(* IEC 61131-3 sources: Word/plc-course/07-timers/labs/solutions, 5 files *)

(* ---- 07-1-star-delta.st ---- *)
(* Lab 07-1: Star-delta starter.
   Module 07 (Timers). REFERENCE SOLUTION - try the lab yourself first.

   Sequence: Start -> main + star contactors on -> after StarTime the star
   contactor opens -> 100 ms dead time -> delta contactor closes.
   Training exercise only: a real starter also has hard-wired electrical and
   mechanical interlocks between the star and delta contactors. *)

PROGRAM StarDelta
  VAR (* I/O *)
    StartPB       AT %IX0.0 : BOOL;  (* Start push-button, NO: TRUE while pressed *)
    StopPB_NC     AT %IX0.1 : BOOL;  (* Stop push-button, NC: TRUE while NOT pressed *)
    OverloadOK_NC AT %IX0.2 : BOOL;  (* Overload relay contact, NC: TRUE while healthy *)
    MainK         AT %QX0.0 : BOOL;  (* Main (line) contactor *)
    StarK         AT %QX0.1 : BOOL;  (* Star contactor *)
    DeltaK        AT %QX0.2 : BOOL;  (* Delta contactor *)
  END_VAR
  VAR (* settings, e.g. written from an HMI *)
    StarTime : TIME := T#5s;         (* how long the motor starts in star *)
  END_VAR
  VAR (* internal *)
    StarTimer : TON;                 (* times the star period *)
    GapTimer  : TON;                 (* changeover dead time, star off -> delta on *)
  END_VAR

  (* 1. Run latch. The main contactor seals itself in. Stop and the overload
        both break the seal, so releasing Stop or resetting the overload relay
        can never restart the motor on its own. *)
  MainK := (StartPB OR MainK) AND StopPB_NC AND OverloadOK_NC;

  (* 2. Star period. The timer runs while the main contactor is on and is
        reset as soon as it drops out, so every new start gets a full star
        period. The timer is called on every scan, never inside an IF. *)
  StarTimer(IN := MainK, PT := StarTime);
  StarK := MainK AND NOT StarTimer.Q;

  (* 3. Changeover gap. StarTimer.Q is TRUE from the scan in which the star
        contactor is switched off, so GapTimer measures how long star has been
        off. Delta may close only after 100 ms, when the star contactor has
        had time to open and its arc to clear. *)
  GapTimer(IN := StarTimer.Q, PT := T#100ms);

  (* 4. Delta, with a software interlock against star as a second line of
        defence (the first line is the hard-wired interlock in the panel). *)
  DeltaK := MainK AND GapTimer.Q AND NOT StarK;
END_PROGRAM

CONFIGURATION Config0
  RESOURCE Res0 ON PLC
    TASK MainTask(INTERVAL := T#10ms, PRIORITY := 0);
    PROGRAM Inst0 WITH MainTask : StarDelta;
  END_RESOURCE
END_CONFIGURATION

(* ---- 07-2-flasher-beacon.st ---- *)
(* Lab 07-2: Flasher beacon with separate on and off times.
   Module 07 (Timers). REFERENCE SOLUTION - try the lab yourself first.

   Two timers that reset each other form an oscillator:
     OnTimer  times the ON phase  (beacon lit while it is timing),
     OffTimer times the OFF phase (started when OnTimer is done).
   When OffTimer is done, OnTimer's IN goes FALSE for one scan. That resets
   both timers and the cycle starts again with a new ON phase. *)

PROGRAM FlasherBeacon
  VAR (* I/O *)
    Enable AT %IX0.0 : BOOL;   (* flash request, e.g. "machine about to start" *)
    Beacon AT %QX0.0 : BOOL;   (* beacon lamp *)
  END_VAR
  VAR (* settings, e.g. written from an HMI *)
    OnTime  : TIME := T#500ms; (* lamp on time *)
    OffTime : TIME := T#1s;    (* lamp off time *)
  END_VAR
  VAR (* internal *)
    OnTimer  : TON;            (* ON phase *)
    OffTimer : TON;            (* OFF phase *)
  END_VAR

  (* ON phase: runs while enabled, until the OFF phase has finished.
     Removing Enable resets it, so the next enable starts with a full
     ON phase. *)
  OnTimer(IN := Enable AND NOT OffTimer.Q, PT := OnTime);

  (* OFF phase: starts when the ON phase is done. *)
  OffTimer(IN := OnTimer.Q, PT := OffTime);

  (* The lamp is lit while enabled and the ON phase is not yet done. *)
  Beacon := Enable AND NOT OnTimer.Q;
END_PROGRAM

CONFIGURATION Config0
  RESOURCE Res0 ON PLC
    TASK MainTask(INTERVAL := T#10ms, PRIORITY := 0);
    PROGRAM Inst0 WITH MainTask : FlasherBeacon;
  END_RESOURCE
END_CONFIGURATION

(* ---- 07-3-feedback-timeout.st ---- *)
(* Lab 07-3: Motor with run-feedback monitoring.
   Module 07 (Timers). REFERENCE SOLUTION - try the lab yourself first.

   Two supervision timers compare what we ASK the motor to do (MotorRun)
   with what it REPORTS (RunFbk):
     - fail to start: no feedback within StartTimeout of the start,
     - feedback lost: feedback was proven, then missing for LossDelay.
   A fault latches, stops the motor, and can be reset only while the run
   command is off, so a reset can never restart the motor by surprise. *)

PROGRAM FeedbackTimeout
  VAR (* I/O *)
    RunCmd    AT %IX0.0 : BOOL;  (* run request (maintained), TRUE = run *)
    RunFbk    AT %IX0.1 : BOOL;  (* running feedback: contactor aux contact or drive "running" *)
    ResetPB   AT %IX0.2 : BOOL;  (* fault reset push-button, NO *)
    MotorRun  AT %QX0.0 : BOOL;  (* contactor coil / drive run command *)
    FaultLamp AT %QX0.1 : BOOL;  (* fault lamp: on while any fault is latched *)
  END_VAR
  VAR (* settings *)
    StartTimeout : TIME := T#3s;     (* time allowed for feedback after a start *)
    LossDelay    : TIME := T#500ms;  (* feedback dropout tolerated while running *)
  END_VAR
  VAR (* alarms for the HMI *)
    FailToStart : BOOL;          (* latched: no feedback after starting *)
    FbkLost     : BOOL;          (* latched: feedback lost while running *)
  END_VAR
  VAR (* internal *)
    Proven     : BOOL;           (* feedback has been seen during this run *)
    StartTimer : TON;            (* supervises the start *)
    LossTimer  : TON;            (* supervises the running motor *)
  END_VAR

  (* 1. "Proven" remembers that feedback arrived during the current run.
        It is cleared whenever the motor is not being commanded, so every new
        start is supervised by the start timer again. MotorRun here is the
        value written at the end of the previous scan. *)
  IF NOT MotorRun THEN
    Proven := FALSE;
  ELSIF RunFbk THEN
    Proven := TRUE;
  END_IF;

  (* 2. Supervision timers. Both are called on every scan; their IN
        conditions decide when they time. *)
  StartTimer(IN := MotorRun AND NOT Proven, PT := StartTimeout);
  LossTimer(IN := MotorRun AND Proven AND NOT RunFbk, PT := LossDelay);

  (* 3. Latch the faults. *)
  IF StartTimer.Q THEN
    FailToStart := TRUE;
  END_IF;
  IF LossTimer.Q THEN
    FbkLost := TRUE;
  END_IF;

  (* 4. Reset, accepted only while the run command is off. *)
  IF ResetPB AND NOT RunCmd THEN
    FailToStart := FALSE;
    FbkLost := FALSE;
  END_IF;

  (* 5. Outputs. *)
  FaultLamp := FailToStart OR FbkLost;
  MotorRun := RunCmd AND NOT FaultLamp;
END_PROGRAM

CONFIGURATION Config0
  RESOURCE Res0 ON PLC
    TASK MainTask(INTERVAL := T#10ms, PRIORITY := 0);
    PROGRAM Inst0 WITH MainTask : FeedbackTimeout;
  END_RESOURCE
END_CONFIGURATION

(* ---- 07-4-run-hours.st ---- *)
(* Lab 07-4: Accumulating run-hours meter.
   Module 07 (Timers). REFERENCE SOLUTION - try the lab yourself first.

   Idea: use a TON purely as a stopwatch. Its ET shows how long the motor has
   been running in the current run. Every scan, add how much ET has grown
   since the previous scan to a small TIME "Fraction", and carry each whole
   second from Fraction into an integer counter. Nothing is thrown away when
   the motor stops, and no time is lost by restarting a short timer every
   second.

   The total lives in a DINT, not a TIME: on many PLCs TIME is a 32-bit
   millisecond count that overflows after about 24.8 days, and a pump can run
   for years. A DINT of seconds lasts about 68 years.

   The TIME arithmetic below (+ and - on TIME values) is standard IEC 61131-3.
   Older code may write the same with ADD_TIME(a, b) and SUB_TIME(a, b). *)

PROGRAM RunHours
  VAR (* I/O *)
    Running    AT %IX0.0 : BOOL;  (* motor running feedback *)
    ResetPB    AT %IX0.1 : BOOL;  (* reset the meter, e.g. after an overhaul (NO) *)
    ServiceDue AT %QX0.0 : BOOL;  (* service-due lamp *)
  END_VAR
  VAR RETAIN (* on a real PLC these must survive a power cut *)
    TotalSeconds : DINT;          (* total running time, whole seconds *)
    Fraction     : TIME;          (* running time not yet counted, below 1 s *)
  END_VAR
  VAR (* display values, recalculated every scan *)
    Hours   : DINT;               (* whole hours *)
    Minutes : DINT;               (* minutes past the whole hour, 0..59 *)
  END_VAR
  VAR (* settings *)
    ServiceHours : DINT := 1000;  (* service interval in running hours *)
  END_VAR
  VAR (* internal *)
    Stopwatch : TON;              (* measures the current run *)
    LastET    : TIME;             (* Stopwatch.ET at the previous scan *)
  END_VAR

  (* 1. Stopwatch. It runs while the motor runs. Its ET would stick at PT, so
        it restarts itself once an hour; that costs two scans an hour
        (0.0006 % with a 10 ms task), which is negligible. *)
  Stopwatch(IN := Running AND NOT Stopwatch.Q, PT := T#1h);

  (* 2. Add the time that has passed since the previous scan. ET only grows
        while the stopwatch is running. When the motor stops (or the stopwatch
        restarts) ET falls back to zero and nothing is added. *)
  IF Stopwatch.ET > LastET THEN
    Fraction := Fraction + (Stopwatch.ET - LastET);
  END_IF;
  LastET := Stopwatch.ET;

  (* 3. Carry whole seconds into the counter. *)
  IF Fraction >= T#1s THEN
    TotalSeconds := TotalSeconds + 1;
    Fraction := Fraction - T#1s;
  END_IF;

  (* 4. Reset: clears the total AND the part-second, and holds both at zero
        while the button is pressed. *)
  IF ResetPB THEN
    TotalSeconds := 0;
    Fraction := T#0s;
  END_IF;

  (* 5. Display values and service reminder. *)
  Hours := TotalSeconds / 3600;
  Minutes := (TotalSeconds MOD 3600) / 60;
  ServiceDue := Hours >= ServiceHours;
END_PROGRAM

CONFIGURATION Config0
  RESOURCE Res0 ON PLC
    TASK MainTask(INTERVAL := T#10ms, PRIORITY := 0);
    PROGRAM Inst0 WITH MainTask : RunHours;
  END_RESOURCE
END_CONFIGURATION

(* ---- 07-5-two-hand-control.st ---- *)
(* Lab 07-5: Two-hand control timing.
   Module 07 (Timers). REFERENCE SOLUTION - try the lab yourself first.

   TRAINING EXERCISE ONLY. A real two-hand control device is a safety function:
   it must use safety-rated buttons (usually one NO and one NC contact each)
   and a safety relay or safety PLC designed to the functional-safety
   standards (Module 20). Never build it from this standard-PLC logic.

   Rules implemented:
     - the stroke runs only while BOTH buttons are held,
     - the second button must follow the first within 500 ms,
     - after any release, BOTH buttons must be released before a new stroke. *)

PROGRAM TwoHandControl
  VAR (* I/O *)
    LeftPB    AT %IX0.0 : BOOL;  (* left palm button, NO: TRUE while pressed *)
    RightPB   AT %IX0.1 : BOOL;  (* right palm button, NO: TRUE while pressed *)
    PressDown AT %QX0.0 : BOOL;  (* press stroke valve *)
  END_VAR
  VAR (* internal *)
    Window : TON;                (* time since the FIRST button was pressed *)
    Ready  : BOOL;               (* both buttons have been released since the last stroke *)
  END_VAR

  (* 1. The synchronisation window starts with whichever button is pressed
        first and resets only when both are released. *)
  Window(IN := LeftPB OR RightPB, PT := T#500ms);

  (* 2. Ready is set only when both buttons are released. It starts FALSE,
        so buttons already held (or tied down) at power-up cannot start a
        stroke. *)
  IF NOT LeftPB AND NOT RightPB THEN
    Ready := TRUE;
  END_IF;

  (* 3. Start: both held, ready, and still inside the window.
        Hold: once running, both held is enough (the window has long expired). *)
  PressDown := LeftPB AND RightPB AND (PressDown OR (Ready AND NOT Window.Q));

  (* 4. A stroke uses up Ready: after any release, both buttons must be
        released before the next stroke. *)
  IF PressDown THEN
    Ready := FALSE;
  END_IF;
END_PROGRAM

CONFIGURATION Config0
  RESOURCE Res0 ON PLC
    TASK MainTask(INTERVAL := T#10ms, PRIORITY := 0);
    PROGRAM Inst0 WITH MainTask : TwoHandControl;
  END_RESOURCE
END_CONFIGURATION
